FUNCTION_BLOCK FlushGritScreens_HMI (* Service Interface Function Block Type *)
  (* Standard: 61499-2 *)
  (* Version 0.0, 6/19/2026, Schneider Electric, template *)
  PACKAGE SE.Nereda;
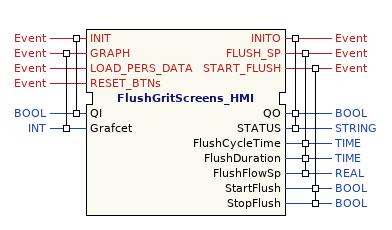
  EVENT_INPUT
    INIT WITH QI;
    GRAPH WITH Grafcet;
    LOAD_PERS_DATA;
    RESET_BTNs;
  END_EVENT
  EVENT_OUTPUT
    INITO WITH QO, STATUS;
    FLUSH_SP WITH FlushCycleTime, FlushDuration, FlushFlowSp;
    START_FLUSH WITH StartFlush, StopFlush;
  END_EVENT
  VAR_INPUT
    QI : BOOL;
    Grafcet : INT;
  END_VAR
  VAR_OUTPUT
    QO : BOOL; (* Event Output Qualifier *)
    STATUS : STRING; (* Service Status *)
    FlushCycleTime : TIME;
    FlushDuration : TIME;
    FlushFlowSp : REAL;
    StartFlush : BOOL;
    StopFlush : BOOL;
  END_VAR
  SERVICE /
    SEQUENCE 
    END_SEQUENCE
  END_SERVICE
END_FUNCTION_BLOCK
